PROGRAM FB_Alarm
  VAR_INPUT
    Fault_in : BOOL;
    Acknowledge : BOOL;
    Alarm_Reset : BOOL;
  END_VAR
  VAR_OUTPUT
    Active : BOOL;
    Latched : BOOL;
  END_VAR
  VAR
    Acknowledged : BOOL;
  END_VAR

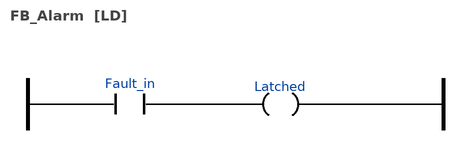
(* LD diagram, written out as Structured Text *)
Latched := Fault_in;
END_PROGRAM
